{attribute 'pack_mode' := '2'}
TYPE ST_In :
STRUCT


  bFastStop         : BIT;  // Fast stop function of NC with mapped input

  {attribute 'hide'}
  b1 : BIT; // hide bit; for future use
  {attribute 'hide'}
  b2 : BIT; // hide bit; for future use
  {attribute 'hide'}
  b3 : BIT; // hide bit; for future use
  {attribute 'hide'}
  b4 : BIT; // hide bit; for future use
  {attribute 'hide'}
  b5 : BIT; // hide bit; for future use
  {attribute 'hide'}
  b6 : BIT;
  {attribute 'hide'}
  b7 : BIT;

  byAxisFuncPara    : BYTE; // additional parameter for Axis Function; e.g. used for AxisIndex on GearIn

  uiAxisFunctionReq : E_AXIS_CTRL; // selected function for axis 

  (* LREAL required by process *)
  rSetPos           : LREAL;
  rSetVelo          : LREAL;
  rOverride         : LREAL;
  rAcc              : LREAL;
  rDec              : LREAL;
  iDirection        : INT;

  {attribute 'hide'}
  w1 : ARRAY[1..3] OF WORD;

END_STRUCT
END_TYPE

(* stored: Version 1.1.0.1, ProductVersion 3.1.4024.12
   DUT ST_In: Id {4dbe302c-d03d-4028-a932-4590e96ac4dc} *)
